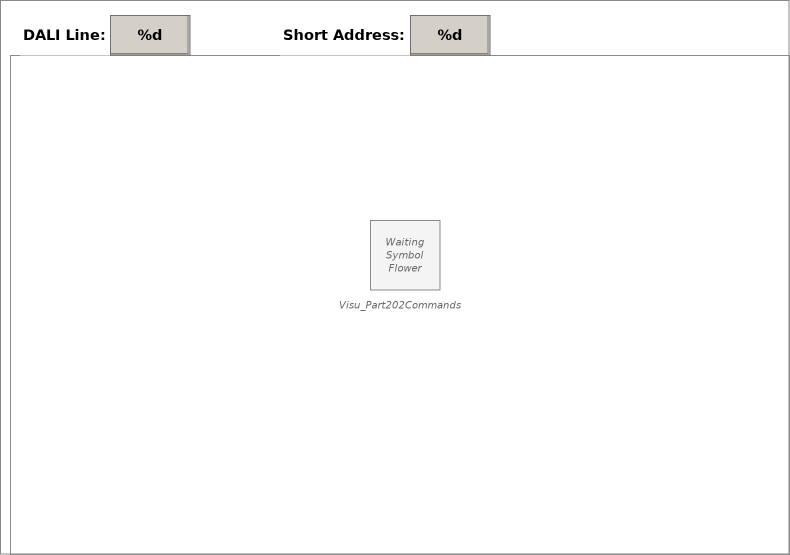
VISUALIZATION Visu_Part202  // 790x555
    TabControl (10,55 780x500)
        shows Visu_Part202Commands()
        shows Visu_Part202Status()
        shows Visu_Part202Parameters()
        [0]: TabTitle=Commands
        [1]: TabTitle=Status
        [2]: TabTitle=Parameters
    Group (280,15 210x40)
        Textfield (0,0 130x40), "Short Address:"
        Button (130,0 80x40), "%d", text variable: DALI_Commissioning.fbPart202Emergency.nAddress
            OnMouseClick: write the text variable via Default, min 0, max 63, title "Insert Short Address"
    Group (20,15 170x40)
        Textfield (0,0 110x40), "DALI Line:"
        Button (90,0 80x40), "%d", text variable: GVL_Internal.nDALILine
            OnMouseClick: write the text variable via Default, min 1, max 10, title "Choose line"
    WaitingSymbolFlower (370,220 70x70), invisible if: DALI_Commissioning.fbPart202Emergency.bHideWaitSymbol
END_VISUALIZATION

(* stored: Version 1.1.0.1, ProductVersion 3.1.4024.12
   Visu Visu_Part202: Id {21862d36-2ce3-434e-aea3-ff61204e05f1} *)
